(* This function evaluates the Turbo ILK logic*)
(* The function switches off the Turbo if the Inlet pressure or the backing Pressure*)
(* are higher than the configured set point*)
FUNCTION F_TurboExtILKLogic_2 : BOOL
VAR_INPUT
	Turbo		:	ST_PTM;
	BackingGauge:	ST_VG;
	InletGauge	:	ST_VG;
	ScrollPump	:	ST_RoughPump;
END_VAR
VAR
END_VAR

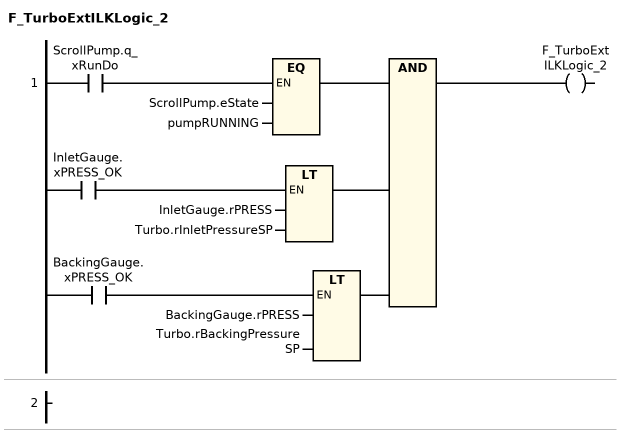
// NETWORK 1
F_TurboExtILKLogic_2 := (ScrollPump.q_xRunDo AND ScrollPump.eState = pumpRUNNING) AND (InletGauge.xPRESS_OK AND InletGauge.rPRESS < Turbo.rInletPressureSP) AND (BackingGauge.xPRESS_OK AND BackingGauge.rPRESS < Turbo.rBackingPressureSP);

// NETWORK 2

END_FUNCTION

(* stored: Version 1.1.0.1, ProductVersion 3.1.4024.3
   POU F_TurboExtILKLogic_2: Id {ed78e581-09e2-43e8-9d0f-45246ab5877a}, SpecialFunc None *)
